TYPE ST_MKS_422 EXTENDS ST_VacuumGauge :
STRUCT
	
	//Ion gauges only
	i_xHvOn	:	BOOL;
	
	// Simulation parameters
	tonIC	:	TON := (PT := T#10S);
END_STRUCT
END_TYPE

(* stored: Version 1.1.0.1, ProductVersion 3.1.4018.5
   DUT ST_MKS_422: Id {e02c8287-6648-4f78-b4be-5219b3c43dad} *)
